// TIA Portal V21 export
DATA_BLOCK "LogoCliente"   // DB6
{ S7_Optimized_Access := 'TRUE' }
// stored: MemoryReserve 100
   VAR RETAIN
      K_LogoCliente_1 : Int := 1;
      K_LogoCliente_2 : Int := 2;
   END_VAR
BEGIN
END_DATA_BLOCK
